// TwinCAT 3 PLC project Tester
// ProgramVersion: 3.1.4026.12
// libraries:
//   Tc2_Standard, * (Beckhoff Automation GmbH)
//   Tc2_System, * (Beckhoff Automation GmbH)
//   Tc2_Utilities, * (Beckhoff Automation GmbH)
// project tree:
//   DUTs/ E_TestEnum.TcDUT, ST_StringForArray.TcDUT, U_EveryType.TcDUT
//   GVLs/ GVL_System.TcGVL
//   / ITest.TcIO, PlcTask.TcTTO
//   POUs/ FB_InterfaceTest.TcPOU, MAIN.TcPOU, FB_TestBlock.TcPOU
// real-time tasks:
//   TASK PlcTask: cycle T#10ms, priority 20, ADS port 350

CONFIGURATION Tester
    RESOURCE PLC ON TwinCAT3
        TASK PlcTask(INTERVAL := T#10ms, PRIORITY := 20);
        PROGRAM MAIN WITH PlcTask : MAIN;
    END_RESOURCE
END_CONFIGURATION

// ---- DUTs/E_TestEnum.TcDUT
{attribute 'qualified_only'}
{attribute 'strict'}
{attribute 'to_string'}
TYPE E_TestEnum :
(
	Idle := 0,
	Starting,
	Running,
	Stopping,
	Pausing,
	Paused,
	Error,
	ErrorResetting
) UINT;
END_TYPE

// ---- DUTs/ST_StringForArray.TcDUT
(*
	Allows direct reading of strings of arrays, inside a structure/function block/program, in a single read from C#
*)
TYPE ST_StringForArray :
STRUCT
	(* String for array *)
	str	: STRING;
END_STRUCT
END_TYPE

// ---- DUTs/U_EveryType.TcDUT
TYPE U_EveryType :
UNION
	(* Boolean *)
	boolean : BOOL;
	(* Integer *)
	integer	: LINT;
	(* Unsigned integer *)
	unsignedInteger : ULINT;
	(* Real number *)
	realNumber : LREAL;
	(* Time *)
	some : TIME;
	(* Date *)
	out : DATE;

END_UNION
END_TYPE

// ---- GVLs/GVL_System.TcGVL
{attribute 'qualified_only'}
{attribute 'NotBlockWritable'}
VAR_GLOBAL
	(* Timestamp for cycle in ISO 8601 format (yyyy-MM-ddTHH:mm:ss.fffZ) *)
	timestamp : STRING(24);
END_VAR

// ---- ITest.TcIO
INTERFACE ITest

METHOD TestMethod : BOOL
VAR_INPUT
END_VAR
END_METHOD

END_INTERFACE

// ---- POUs/MAIN.TcPOU
{attribute 'NotBlockWritable'}
PROGRAM MAIN
VAR
	(* Boolean *)
	boolean : BOOL;
	(* Integer *)
	integer	: LINT;
	(* Unsigned integer *)
	unsignedInteger : ULINT;
	(* Real number *)
	realNumber : REAL;
	(* Text (80 characters) *)
	text : STRING;
	(* Time *)
	some : TIME;
	(* Date *)
	out : DATE;
	(* Array of text (80 characters each) *)
	localStringArray : ARRAY [0..10] OF STRING;

	(* Enumeration *)
	state : E_TestEnum := E_TestEnum.Idle;
	
	(* Function Block *)
	testBlock	: FB_TestBlock;
	(* Function Block using Interface *)
	testInterface : FB_InterfaceTest;
	
	(* Indirect array of strings *)
	easyToReadString : ARRAY [0..10] OF ST_StringForArray;
	
	(* Multidiminsional array *)
	ArrayArray : ARRAY [0..10,0..10] OF BOOL;
	
	(* Array of array *)
	ArrayOfArray : ARRAY [0..10] OF ARRAY [0..10] OF ULINT;

	(* Union *)
	item : U_EveryType;
	
	(* Windows time *)
	{attribute 'NotBlockWritable'}
	fbTime   : FB_LocalSystemTime := ( bEnable := TRUE, dwCycle := 1 );
	(* Windows time zone *)
	{attribute 'NotBlockWritable'}
	fbTimeZone : FB_GetTimeZoneInformation := (bExecute := TRUE);
	(* Converts local Windows time to UTC *)
	{attribute 'NotBlockWritable'}
	fbToUTC : FB_TzSpecificLocalTimeToSystemTime;
END_VAR

VAR PERSISTENT
	testCallDelayTime : TIME := T#5s;
END_VAR

(* Hidden gem, a quick/cheap way to get a timestamp for log messages for this PLC cycle *)
fbTime();
fbTimeZone();
IF fbtime.bValid AND NOT fbTimeZone.bBusy THEN
	(* Once the time and time zone are valid, convert system time to UTC *)
	fbToUTC(in := fbTime.systemTime,
			tzInfo := fbTimeZone.tzInfo);
			
	(* Convert the UTC system time into the ISO8601 format for UTC, fixing the timezone bug in Beckhoff's code *)
	GVL_System.timestamp := SystemTime_To_ISO8601(systemTime := fbToUTC.out,
												  nBias := 0,
												  bUTC := TRUE,
												  nPrecision := 3);
	GVL_System.timestamp := REPLACE(GVL_System.timestamp, 'Z',1,24);
END_IF

(* Run the test function block *)
testBlock(interfaceTest := testInterface, delayUpdates := testCallDelayTime);

(* Update the union with the new value *)
item.integer := testBlock.callCount;

END_PROGRAM

// ---- POUs/FB_TestBlock.TcPOU
{attribute 'NotBlockWritable'}
FUNCTION_BLOCK FB_TestBlock
VAR_INPUT
	(* Time between calls to the interface *)
	delayUpdates : TIME;
	(* Interface to call when time it over *)
	interfaceTest : ITest;
END_VAR

VAR_OUTPUT
	(* Counter of calls made *)
	callCount : UINT;
END_VAR

VAR
	(* Counter of calls made with a return of TRUE *)
	trueCallCount : UINT;
	(* Timer for the call *)
	{attribute 'ReadOnly'}
	callTimer : TON;
	(* Reference to another Function Block of the same time *)
	selfTypeReference : REFERENCE TO FB_TestBlock;
END_VAR

(* Call the interface every delayUpdates time *)
callTimer(IN := TRUE, PT := delayUpdates);
IF callTimer.Q THEN
	(* Reset the timer and increase the call count *)
	callTimer(IN := FALSE);
	callCount := callCount + 1;
	
	(* Protect against a bad interface and call the method, increasing trueCallCount if true *)
	IF interfaceTest <> 0 THEN
		IF interfaceTest.TestMethod() THEN
			trueCallCount := trueCallCount + 1;
		END_IF
	END_IF
END_IF

END_FUNCTION_BLOCK

// ---- POUs/FB_InterfaceTest.TcPOU
(*
	Function block to assign to an ITest interface
*)
{attribute 'NotBlockWritable'}
FUNCTION_BLOCK FB_InterfaceTest IMPLEMENTS ITest
VAR
	(* Last Value *)
	oldValue : BOOL;
END_VAR

(*
	Test method for the ITest interface
*)
METHOD TestMethod : BOOL	(* Inverted value since last call *)
(* Return the inverted old value and save the inverted value as the new old value *)
TestMethod := NOT oldValue;
oldValue := TestMethod;
END_METHOD

END_FUNCTION_BLOCK
